// TIA Portal V17 export
// export: Created 2025-03-05T08:03:15.5242576Z, ExportSetting WithDefaults, DisplayName Totally Integrated Automation Portal, DisplayVersion V17 Update 8, DisplayName TIA Portal Openness, DisplayVersion V17 Update 8, DisplayName TIA Portal Version Control Interface, DisplayVersion V17, DisplayName SINAMICS Startdrive Advanced, DisplayVersion V17 SP2, DisplayName SINAMICS Startdrive G110M, G120, G120C, G120D, G120P, G115D, DisplayVersion V17 SP2, DisplayName SINAMICS Startdrive G130, G150, S120, S150, SINAMICS MV, S210, DisplayVersion V17 SP2, DisplayName STEP 7 Professional, DisplayVersion V17 Update 8, DisplayName SINUMERIK ONE STEP 7 Toolbox, DisplayVersion V17 Update 12, DisplayName SINUMERIK 840D sl STEP 7 Toolbox, DisplayVersion V17 Update 12, DisplayName STEP 7 Safety, DisplayVersion V17 Update 6, DisplayName WinCC Advanced, DisplayVersion V17 Update 8
FUNCTION_BLOCK "FB22500_PRESSURE_CONTROL_REGTONIC"   // FB22500, LAD
{ S7_Optimized_Access := 'FALSE' }
VERSION : 0.1
// stored: AutoNumber false, IsIECCheckEnabled false, SetENOAutomatically false, UDAEnableTagReadback false
   VAR_INPUT
      CONTROL_ON_DELAYED : Bool;   // CONTROL ON DELAYED
      PNEUMATIC_CONDITIONS : Bool;   // PNEUMATIC CONDITIONS
      FEEDER_NOT_READY_FAULT : Bool;   // FEEDER NOT READY FAULT
      PRESSURIZE_VALVE_FEEDBACK : Bool;   // PRESSURIZE VALVE FEEDBACK
      START_PROGRAM_REQUEST : Bool;   // START PROGRAM REQUEST
      START_MANUAL_REQUEST : Bool;   // START MANUAL REQUEST
      START_SEMI_REQUEST : Bool;   // START SEMI REQUEST
      START_AUTO_REQUEST : Bool;   // START AUTO REQUEST
      STOP_PROGRAM_REQUEST : Bool;   // STOP PROGRAM REQUEST
      STOP_MANUAL_REQUEST : Bool;   // STOP MANUAL REQUEST
      STOP_SEMI_REQUEST : Bool;   // STOP SEMI REQUEST
      STOP_AUTO_REQUEST : Bool;   // STOP AUTO REQUEST
      ACTUAL_PRESSURE : Real;   // ACTUAL PRESSURE
      PRESSURE_SETPOINT_AUTO : Real;   // PRESSURE SETPOINT
   END_VAR
   VAR_OUTPUT
      PRESSURE_CONTROL_VALUE : Int;   // PRESSURE CONTROL VALUE
      SIMULTANEITY_ALARM : Bool;   // SIMULTANEITY ALARM
      TIME_EXCEEDED_ALARM : Bool;   // TIME EXCEEDED ALARM
      SWITCH_ON_ALARM : Bool;   // SWITCH ON ALARM
      SWITCH_OFF_ALARM : Bool;   // SWITCH OFF ALARM
   END_VAR
   VAR_IN_OUT
      DB_PID : PID_Compact;
   END_VAR
   VAR DB_SPECIFIC
      DATA_STANDARD : "GENERAL_DATA_START_STOP";
      START_STOP_HMI { S7_SetPoint := 'True'} : "HMI_DATA_START_STOP";
      INPUT_SETINGS : Struct
         UNIT_NUMBER : Int;
         HOPPER_NUMBER : Int;
      END_STRUCT;
      DATA_HMI : Struct
         PRESSURE_SETPOINT_VALUE : Real;
      END_STRUCT;
      ALARM_SETINGS : Struct
         TIMER_SIMULTANEITY : TON_TIME;   // SIMULTANEITY TIMER
         TIMER_TIME_EXCEEDED { S7_SetPoint := 'True'} : TON_TIME;
      END_STRUCT;
      SETPOINT_PRESSURE : Real;
      CONTROL_PRESSURE_OUTPUT : Int;
   END_VAR
   VAR_TEMP
      DB_NUMBER : DInt;
      RETVAL : Int;
   END_VAR
   // ALARM_SETINGS.TIMER_SIMULTANEITY.PT := T#100ms;
   // ALARM_SETINGS.TIMER_TIME_EXCEEDED.PT := T#4s;
   VAR_TEMP   // added for the SCL form of the ladder/FBD networks
      _w1 : Bool;
      _w2 : Bool;
   END_VAR
BEGIN

NETWORK
TITLE = READ INSTANCE DB NUMBER
      L     DINO;
      +     10#800000;
      T     #DB_NUMBER;



REGION Network 2: GENERAL CONDITIONS START
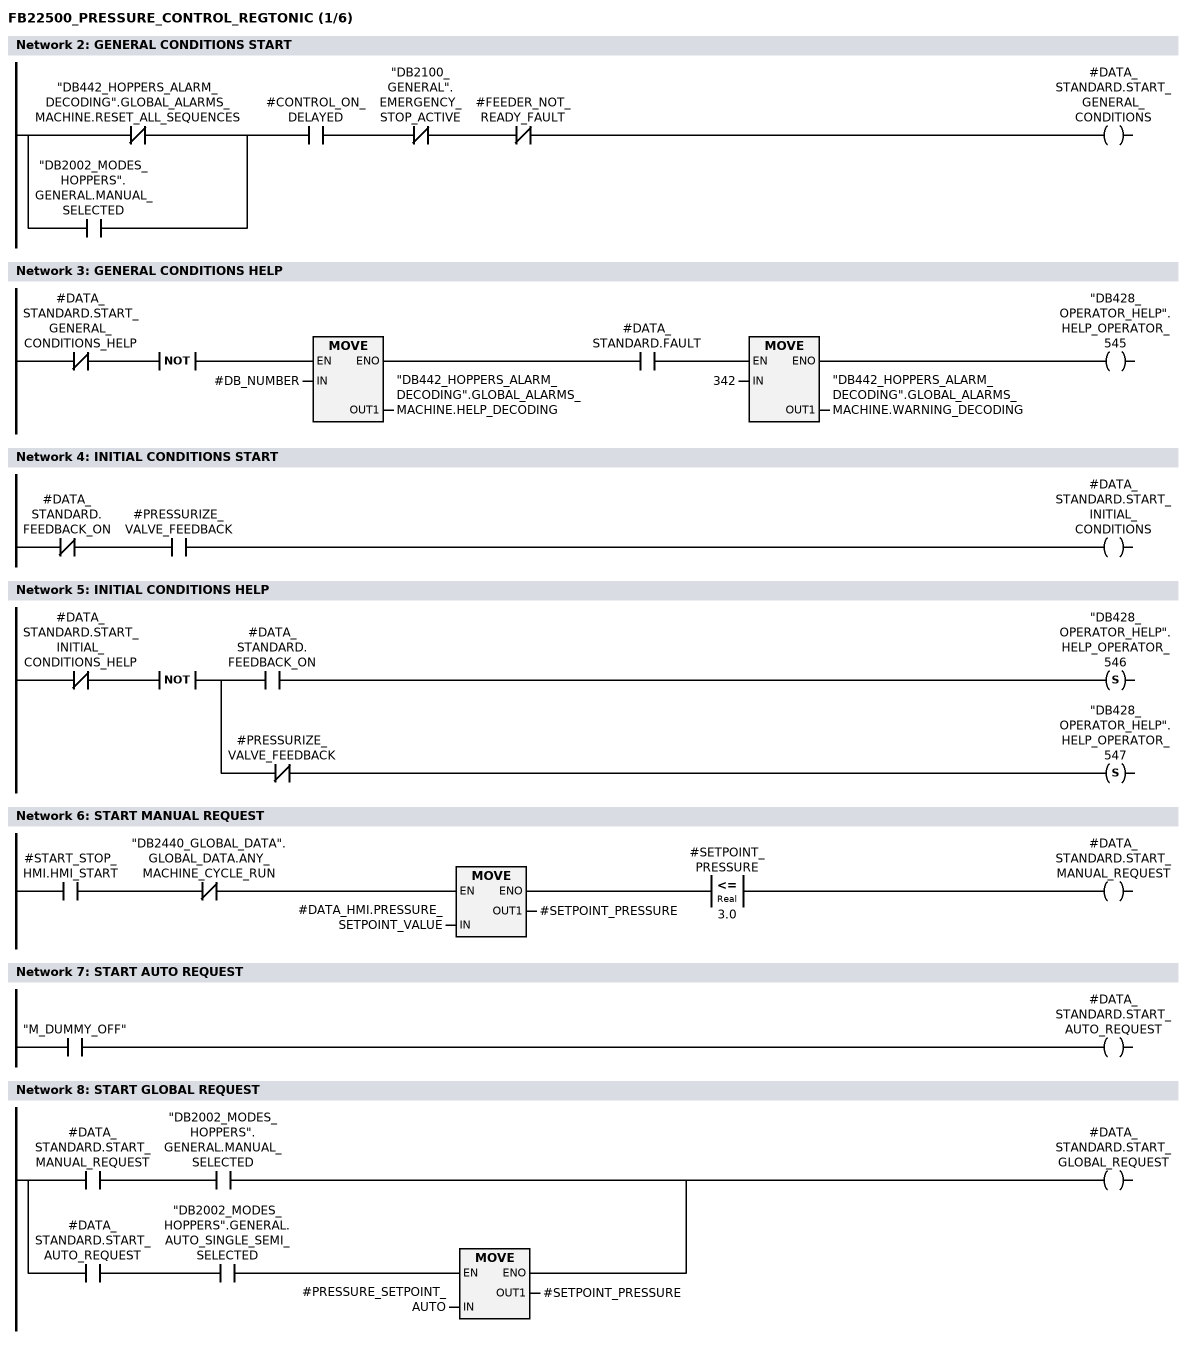
   RUNG wire#powerrail
      I_Contact( "DB442_HOPPERS_ALARM_DECODING".GLOBAL_ALARMS_MACHINE.RESET_ALL_SEQUENCES )
      wire#w1
      Contact( #CONTROL_ON_DELAYED )
      I_Contact( "DB2100_GENERAL".EMERGENCY_STOP_ACTIVE )
      I_Contact( #FEEDER_NOT_READY_FAULT )
      Coil( #DATA_STANDARD.START_GENERAL_CONDITIONS )
   END_RUNG
   RUNG wire#powerrail
      Contact( "DB2002_MODES_HOPPERS".GENERAL.MANUAL_SELECTED )
   END_RUNG wire#w1
   // the same network as SCL:
   #DATA_STANDARD.START_GENERAL_CONDITIONS := (NOT "DB442_HOPPERS_ALARM_DECODING".GLOBAL_ALARMS_MACHINE.RESET_ALL_SEQUENCES OR "DB2002_MODES_HOPPERS".GENERAL.MANUAL_SELECTED) AND #CONTROL_ON_DELAYED AND NOT "DB2100_GENERAL".EMERGENCY_STOP_ACTIVE AND NOT #FEEDER_NOT_READY_FAULT;
END_REGION

REGION Network 3: GENERAL CONDITIONS HELP
   RUNG wire#powerrail
      I_Contact( #DATA_STANDARD.START_GENERAL_CONDITIONS_HELP )
      Not()
      Move(in := #DB_NUMBER, out1 => "DB442_HOPPERS_ALARM_DECODING".GLOBAL_ALARMS_MACHINE.HELP_DECODING)
      Contact( #DATA_STANDARD.FAULT )
      Move(in := 342, out1 => "DB442_HOPPERS_ALARM_DECODING".GLOBAL_ALARMS_MACHINE.WARNING_DECODING)
      Coil( "DB428_OPERATOR_HELP".HELP_OPERATOR_545 )
   END_RUNG
   // the same network as SCL:
   #_w1 := NOT (NOT #DATA_STANDARD.START_GENERAL_CONDITIONS_HELP);
   IF #_w1 THEN "DB442_HOPPERS_ALARM_DECODING".GLOBAL_ALARMS_MACHINE.HELP_DECODING := #DB_NUMBER; END_IF;
   #_w2 := #_w1 AND #DATA_STANDARD.FAULT;
   IF #_w2 THEN "DB442_HOPPERS_ALARM_DECODING".GLOBAL_ALARMS_MACHINE.WARNING_DECODING := 342; END_IF;
   "DB428_OPERATOR_HELP".HELP_OPERATOR_545 := #_w2;
END_REGION

REGION Network 4: INITIAL CONDITIONS START
   RUNG wire#powerrail
      I_Contact( #DATA_STANDARD.FEEDBACK_ON )
      Contact( #PRESSURIZE_VALVE_FEEDBACK )
      Coil( #DATA_STANDARD.START_INITIAL_CONDITIONS )
   END_RUNG
   // the same network as SCL:
   #DATA_STANDARD.START_INITIAL_CONDITIONS := NOT #DATA_STANDARD.FEEDBACK_ON AND #PRESSURIZE_VALVE_FEEDBACK;
END_REGION

REGION Network 5: INITIAL CONDITIONS HELP
   RUNG wire#powerrail
      I_Contact( #DATA_STANDARD.START_INITIAL_CONDITIONS_HELP )
      Not()
      wire#w1
      Contact( #DATA_STANDARD.FEEDBACK_ON )
      S_Coil( "DB428_OPERATOR_HELP".HELP_OPERATOR_546 )
   END_RUNG
   RUNG wire#w1
      I_Contact( #PRESSURIZE_VALVE_FEEDBACK )
      S_Coil( "DB428_OPERATOR_HELP".HELP_OPERATOR_547 )
   END_RUNG
   // the same network as SCL:
   #_w1 := NOT (NOT #DATA_STANDARD.START_INITIAL_CONDITIONS_HELP);
   IF #_w1 AND #DATA_STANDARD.FEEDBACK_ON THEN "DB428_OPERATOR_HELP".HELP_OPERATOR_546 := TRUE; END_IF;
   IF #_w1 AND NOT #PRESSURIZE_VALVE_FEEDBACK THEN "DB428_OPERATOR_HELP".HELP_OPERATOR_547 := TRUE; END_IF;
END_REGION

REGION Network 6: START MANUAL REQUEST
   RUNG wire#powerrail
      Contact( #START_STOP_HMI.HMI_START )
      I_Contact( "DB2440_GLOBAL_DATA".GLOBAL_DATA.ANY_MACHINE_CYCLE_RUN )
      Move(in := #DATA_HMI.PRESSURE_SETPOINT_VALUE, out1 => #SETPOINT_PRESSURE)
      { S7_Templates := "SrcType := Real" } LE_Contact(in1 := #SETPOINT_PRESSURE, in2 := 3.0)
      Coil( #DATA_STANDARD.START_MANUAL_REQUEST )
   END_RUNG
   // the same network as SCL:
   #_w1 := #START_STOP_HMI.HMI_START AND NOT "DB2440_GLOBAL_DATA".GLOBAL_DATA.ANY_MACHINE_CYCLE_RUN;
   IF #_w1 THEN #SETPOINT_PRESSURE := #DATA_HMI.PRESSURE_SETPOINT_VALUE; END_IF;
   #DATA_STANDARD.START_MANUAL_REQUEST := #_w1 AND (#SETPOINT_PRESSURE <= 3.0);
END_REGION

REGION Network 7: START AUTO REQUEST
   RUNG wire#powerrail
      Contact( "M_DUMMY_OFF" )
      Coil( #DATA_STANDARD.START_AUTO_REQUEST )
   END_RUNG
   // the same network as SCL:
   #DATA_STANDARD.START_AUTO_REQUEST := "M_DUMMY_OFF";
END_REGION

REGION Network 8: START GLOBAL REQUEST
   RUNG wire#powerrail
      Contact( #DATA_STANDARD.START_MANUAL_REQUEST )
      Contact( "DB2002_MODES_HOPPERS".GENERAL.MANUAL_SELECTED )
      wire#w1
      Coil( #DATA_STANDARD.START_GLOBAL_REQUEST )
   END_RUNG
   RUNG wire#powerrail
      Contact( #DATA_STANDARD.START_AUTO_REQUEST )
      Contact( "DB2002_MODES_HOPPERS".GENERAL.AUTO_SINGLE_SEMI_SELECTED )
      Move(in := #PRESSURE_SETPOINT_AUTO, out1 => #SETPOINT_PRESSURE)
   END_RUNG wire#w1
   // the same network as SCL:
   #_w1 := #DATA_STANDARD.START_AUTO_REQUEST AND "DB2002_MODES_HOPPERS".GENERAL.AUTO_SINGLE_SEMI_SELECTED;
   IF #_w1 THEN #SETPOINT_PRESSURE := #PRESSURE_SETPOINT_AUTO; END_IF;
   #DATA_STANDARD.START_GLOBAL_REQUEST := (#DATA_STANDARD.START_MANUAL_REQUEST AND "DB2002_MODES_HOPPERS".GENERAL.MANUAL_SELECTED) OR #_w1;
END_REGION

REGION Network 9: START COMMAND
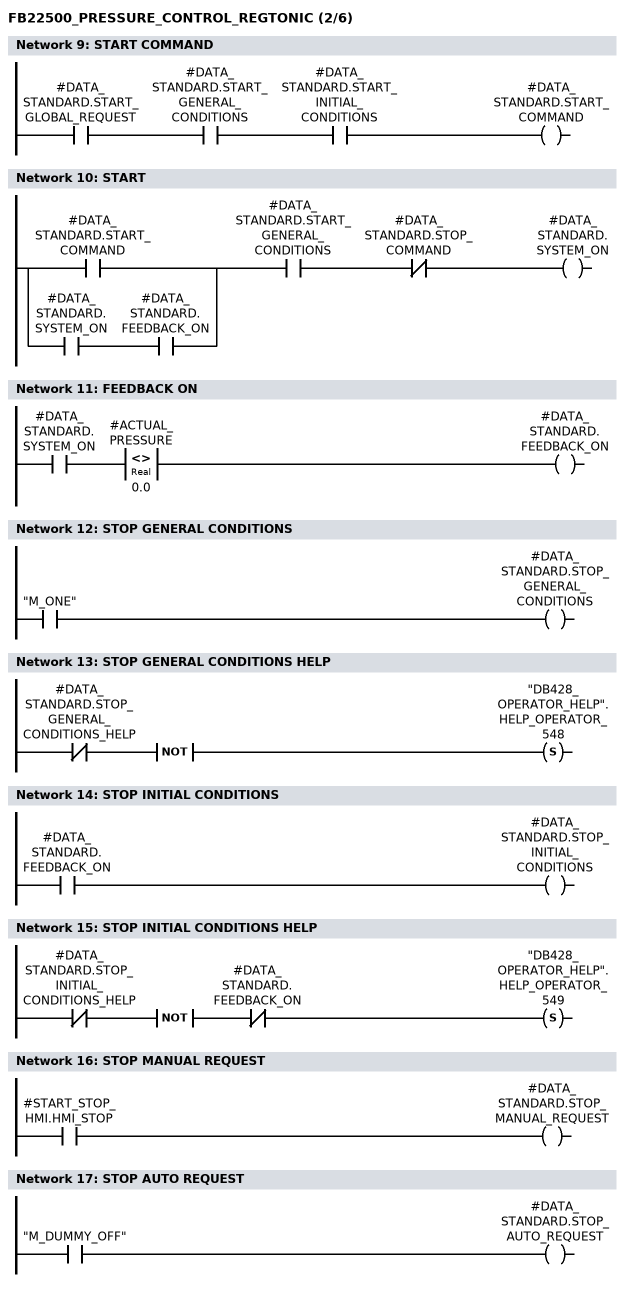
   RUNG wire#powerrail
      Contact( #DATA_STANDARD.START_GLOBAL_REQUEST )
      Contact( #DATA_STANDARD.START_GENERAL_CONDITIONS )
      Contact( #DATA_STANDARD.START_INITIAL_CONDITIONS )
      Coil( #DATA_STANDARD.START_COMMAND )
   END_RUNG
   // the same network as SCL:
   #DATA_STANDARD.START_COMMAND := #DATA_STANDARD.START_GLOBAL_REQUEST AND #DATA_STANDARD.START_GENERAL_CONDITIONS AND #DATA_STANDARD.START_INITIAL_CONDITIONS;
END_REGION

REGION Network 10: START
   RUNG wire#powerrail
      Contact( #DATA_STANDARD.START_COMMAND )
      wire#w1
      Contact( #DATA_STANDARD.START_GENERAL_CONDITIONS )
      I_Contact( #DATA_STANDARD.STOP_COMMAND )
      Coil( #DATA_STANDARD.SYSTEM_ON )
   END_RUNG
   RUNG wire#powerrail
      Contact( #DATA_STANDARD.SYSTEM_ON )
      Contact( #DATA_STANDARD.FEEDBACK_ON )
   END_RUNG wire#w1
   // the same network as SCL:
   #DATA_STANDARD.SYSTEM_ON := (#DATA_STANDARD.START_COMMAND OR (#DATA_STANDARD.SYSTEM_ON AND #DATA_STANDARD.FEEDBACK_ON)) AND #DATA_STANDARD.START_GENERAL_CONDITIONS AND NOT #DATA_STANDARD.STOP_COMMAND;
END_REGION

REGION Network 11: FEEDBACK ON
   RUNG wire#powerrail
      Contact( #DATA_STANDARD.SYSTEM_ON )
      { S7_Templates := "SrcType := Real" } NE_Contact(in1 := #ACTUAL_PRESSURE, in2 := 0.0)
      Coil( #DATA_STANDARD.FEEDBACK_ON )
   END_RUNG
   // the same network as SCL:
   #DATA_STANDARD.FEEDBACK_ON := #DATA_STANDARD.SYSTEM_ON AND (#ACTUAL_PRESSURE <> 0.0);
END_REGION

REGION Network 12: STOP GENERAL CONDITIONS
   RUNG wire#powerrail
      Contact( "M_ONE" )
      Coil( #DATA_STANDARD.STOP_GENERAL_CONDITIONS )
   END_RUNG
   // the same network as SCL:
   #DATA_STANDARD.STOP_GENERAL_CONDITIONS := "M_ONE";
END_REGION

REGION Network 13: STOP GENERAL CONDITIONS HELP
   RUNG wire#powerrail
      I_Contact( #DATA_STANDARD.STOP_GENERAL_CONDITIONS_HELP )
      Not()
      S_Coil( "DB428_OPERATOR_HELP".HELP_OPERATOR_548 )
   END_RUNG
   // the same network as SCL:
   IF NOT (NOT #DATA_STANDARD.STOP_GENERAL_CONDITIONS_HELP) THEN
       "DB428_OPERATOR_HELP".HELP_OPERATOR_548 := TRUE;
   END_IF;
END_REGION

REGION Network 14: STOP INITIAL CONDITIONS
   RUNG wire#powerrail
      Contact( #DATA_STANDARD.FEEDBACK_ON )
      Coil( #DATA_STANDARD.STOP_INITIAL_CONDITIONS )
   END_RUNG
   // the same network as SCL:
   #DATA_STANDARD.STOP_INITIAL_CONDITIONS := #DATA_STANDARD.FEEDBACK_ON;
END_REGION

REGION Network 15: STOP INITIAL CONDITIONS HELP
   RUNG wire#powerrail
      I_Contact( #DATA_STANDARD.STOP_INITIAL_CONDITIONS_HELP )
      Not()
      I_Contact( #DATA_STANDARD.FEEDBACK_ON )
      S_Coil( "DB428_OPERATOR_HELP".HELP_OPERATOR_549 )
   END_RUNG
   // the same network as SCL:
   IF NOT (NOT #DATA_STANDARD.STOP_INITIAL_CONDITIONS_HELP) AND NOT #DATA_STANDARD.FEEDBACK_ON THEN
       "DB428_OPERATOR_HELP".HELP_OPERATOR_549 := TRUE;
   END_IF;
END_REGION

REGION Network 16: STOP MANUAL REQUEST
   RUNG wire#powerrail
      Contact( #START_STOP_HMI.HMI_STOP )
      Coil( #DATA_STANDARD.STOP_MANUAL_REQUEST )
   END_RUNG
   // the same network as SCL:
   #DATA_STANDARD.STOP_MANUAL_REQUEST := #START_STOP_HMI.HMI_STOP;
END_REGION

REGION Network 17: STOP AUTO REQUEST
   RUNG wire#powerrail
      Contact( "M_DUMMY_OFF" )
      Coil( #DATA_STANDARD.STOP_AUTO_REQUEST )
   END_RUNG
   // the same network as SCL:
   #DATA_STANDARD.STOP_AUTO_REQUEST := "M_DUMMY_OFF";
END_REGION

REGION Network 18: STOP GLOBAL REQUEST
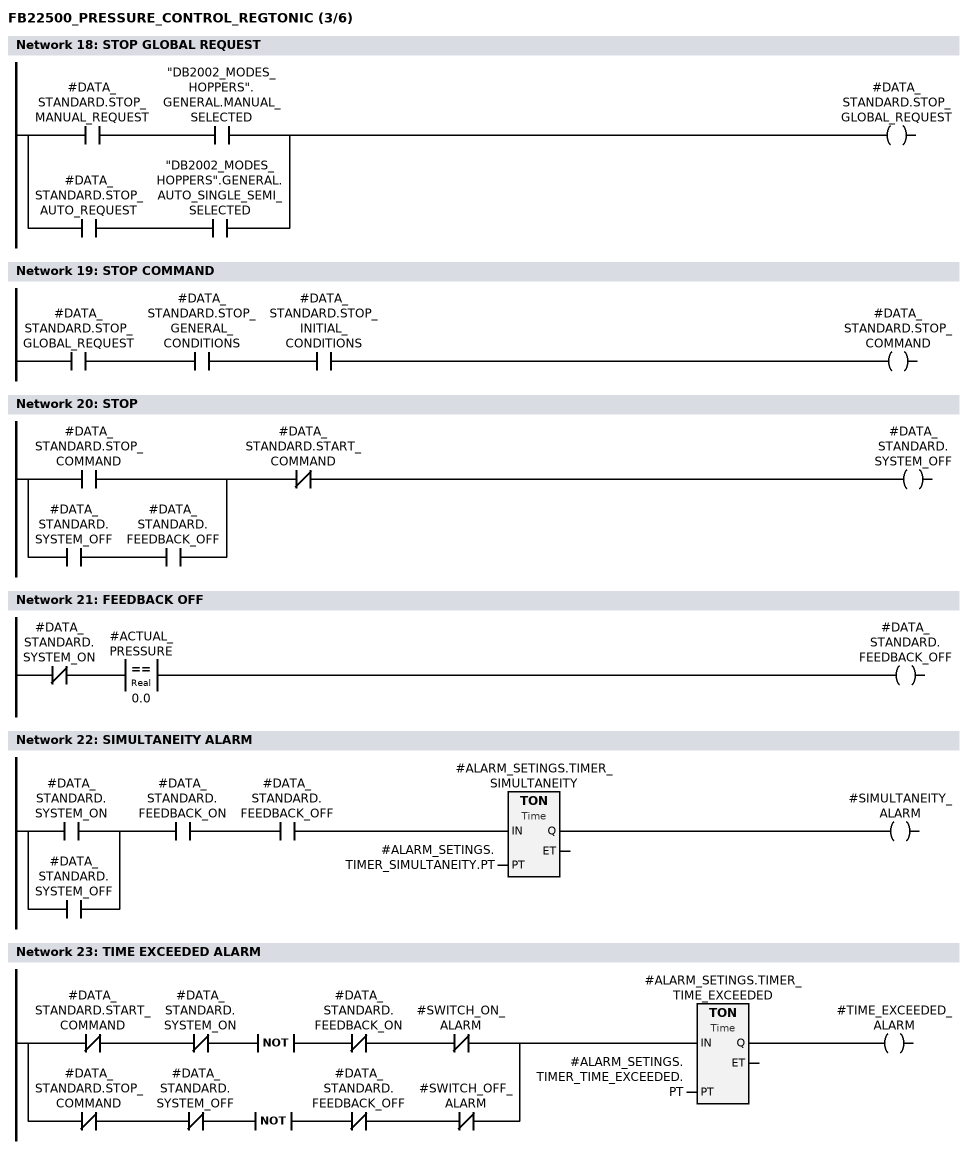
   RUNG wire#powerrail
      Contact( #DATA_STANDARD.STOP_MANUAL_REQUEST )
      Contact( "DB2002_MODES_HOPPERS".GENERAL.MANUAL_SELECTED )
      wire#w1
      Coil( #DATA_STANDARD.STOP_GLOBAL_REQUEST )
   END_RUNG
   RUNG wire#powerrail
      Contact( #DATA_STANDARD.STOP_AUTO_REQUEST )
      Contact( "DB2002_MODES_HOPPERS".GENERAL.AUTO_SINGLE_SEMI_SELECTED )
   END_RUNG wire#w1
   // the same network as SCL:
   #DATA_STANDARD.STOP_GLOBAL_REQUEST := (#DATA_STANDARD.STOP_MANUAL_REQUEST AND "DB2002_MODES_HOPPERS".GENERAL.MANUAL_SELECTED) OR (#DATA_STANDARD.STOP_AUTO_REQUEST AND "DB2002_MODES_HOPPERS".GENERAL.AUTO_SINGLE_SEMI_SELECTED);
END_REGION

REGION Network 19: STOP COMMAND
   RUNG wire#powerrail
      Contact( #DATA_STANDARD.STOP_GLOBAL_REQUEST )
      Contact( #DATA_STANDARD.STOP_GENERAL_CONDITIONS )
      Contact( #DATA_STANDARD.STOP_INITIAL_CONDITIONS )
      Coil( #DATA_STANDARD.STOP_COMMAND )
   END_RUNG
   // the same network as SCL:
   #DATA_STANDARD.STOP_COMMAND := #DATA_STANDARD.STOP_GLOBAL_REQUEST AND #DATA_STANDARD.STOP_GENERAL_CONDITIONS AND #DATA_STANDARD.STOP_INITIAL_CONDITIONS;
END_REGION

REGION Network 20: STOP
   RUNG wire#powerrail
      Contact( #DATA_STANDARD.STOP_COMMAND )
      wire#w1
      I_Contact( #DATA_STANDARD.START_COMMAND )
      Coil( #DATA_STANDARD.SYSTEM_OFF )
   END_RUNG
   RUNG wire#powerrail
      Contact( #DATA_STANDARD.SYSTEM_OFF )
      Contact( #DATA_STANDARD.FEEDBACK_OFF )
   END_RUNG wire#w1
   // the same network as SCL:
   #DATA_STANDARD.SYSTEM_OFF := (#DATA_STANDARD.STOP_COMMAND OR (#DATA_STANDARD.SYSTEM_OFF AND #DATA_STANDARD.FEEDBACK_OFF)) AND NOT #DATA_STANDARD.START_COMMAND;
END_REGION

REGION Network 21: FEEDBACK OFF
   RUNG wire#powerrail
      I_Contact( #DATA_STANDARD.SYSTEM_ON )
      { S7_Templates := "SrcType := Real" } EQ_Contact(in1 := #ACTUAL_PRESSURE, in2 := 0.0)
      Coil( #DATA_STANDARD.FEEDBACK_OFF )
   END_RUNG
   // the same network as SCL:
   #DATA_STANDARD.FEEDBACK_OFF := NOT #DATA_STANDARD.SYSTEM_ON AND (#ACTUAL_PRESSURE = 0.0);
END_REGION

REGION Network 22: SIMULTANEITY ALARM
   RUNG wire#powerrail
      Contact( #DATA_STANDARD.SYSTEM_ON )
      wire#w1
      Contact( #DATA_STANDARD.FEEDBACK_ON )
      Contact( #DATA_STANDARD.FEEDBACK_OFF )
      { S7_Templates := "time_type := Time" } #ALARM_SETINGS.TIMER_SIMULTANEITY.TON(pt := #ALARM_SETINGS.TIMER_SIMULTANEITY.PT, et =>)
      Coil( #SIMULTANEITY_ALARM )
   END_RUNG
   RUNG wire#powerrail
      Contact( #DATA_STANDARD.SYSTEM_OFF )
   END_RUNG wire#w1
   // the same network as SCL:
   #ALARM_SETINGS.TIMER_SIMULTANEITY.TON(IN := (#DATA_STANDARD.SYSTEM_ON OR #DATA_STANDARD.SYSTEM_OFF) AND #DATA_STANDARD.FEEDBACK_ON AND #DATA_STANDARD.FEEDBACK_OFF,
                           PT := #ALARM_SETINGS.TIMER_SIMULTANEITY.PT);
   #SIMULTANEITY_ALARM := #ALARM_SETINGS.TIMER_SIMULTANEITY.Q;
END_REGION

REGION Network 23: TIME EXCEEDED ALARM
   RUNG wire#powerrail
      I_Contact( #DATA_STANDARD.START_COMMAND )
      I_Contact( #DATA_STANDARD.SYSTEM_ON )
      Not()
      I_Contact( #DATA_STANDARD.FEEDBACK_ON )
      I_Contact( #SWITCH_ON_ALARM )
      wire#w1
      { S7_Templates := "time_type := Time" } #ALARM_SETINGS.TIMER_TIME_EXCEEDED.TON(pt := #ALARM_SETINGS.TIMER_TIME_EXCEEDED.PT, et =>)
      Coil( #TIME_EXCEEDED_ALARM )
   END_RUNG
   RUNG wire#powerrail
      I_Contact( #DATA_STANDARD.STOP_COMMAND )
      I_Contact( #DATA_STANDARD.SYSTEM_OFF )
      Not()
      I_Contact( #DATA_STANDARD.FEEDBACK_OFF )
      I_Contact( #SWITCH_OFF_ALARM )
   END_RUNG wire#w1
   // the same network as SCL:
   #ALARM_SETINGS.TIMER_TIME_EXCEEDED.TON(IN := (NOT (NOT #DATA_STANDARD.START_COMMAND AND NOT #DATA_STANDARD.SYSTEM_ON) AND NOT #DATA_STANDARD.FEEDBACK_ON AND NOT #SWITCH_ON_ALARM) OR (NOT (NOT #DATA_STANDARD.STOP_COMMAND AND NOT #DATA_STANDARD.SYSTEM_OFF) AND NOT #DATA_STANDARD.FEEDBACK_OFF AND NOT #SWITCH_OFF_ALARM),
                           PT := #ALARM_SETINGS.TIMER_TIME_EXCEEDED.PT);
   #TIME_EXCEEDED_ALARM := #ALARM_SETINGS.TIMER_TIME_EXCEEDED.Q;
END_REGION

REGION Network 24: SWITCH ON ALARM
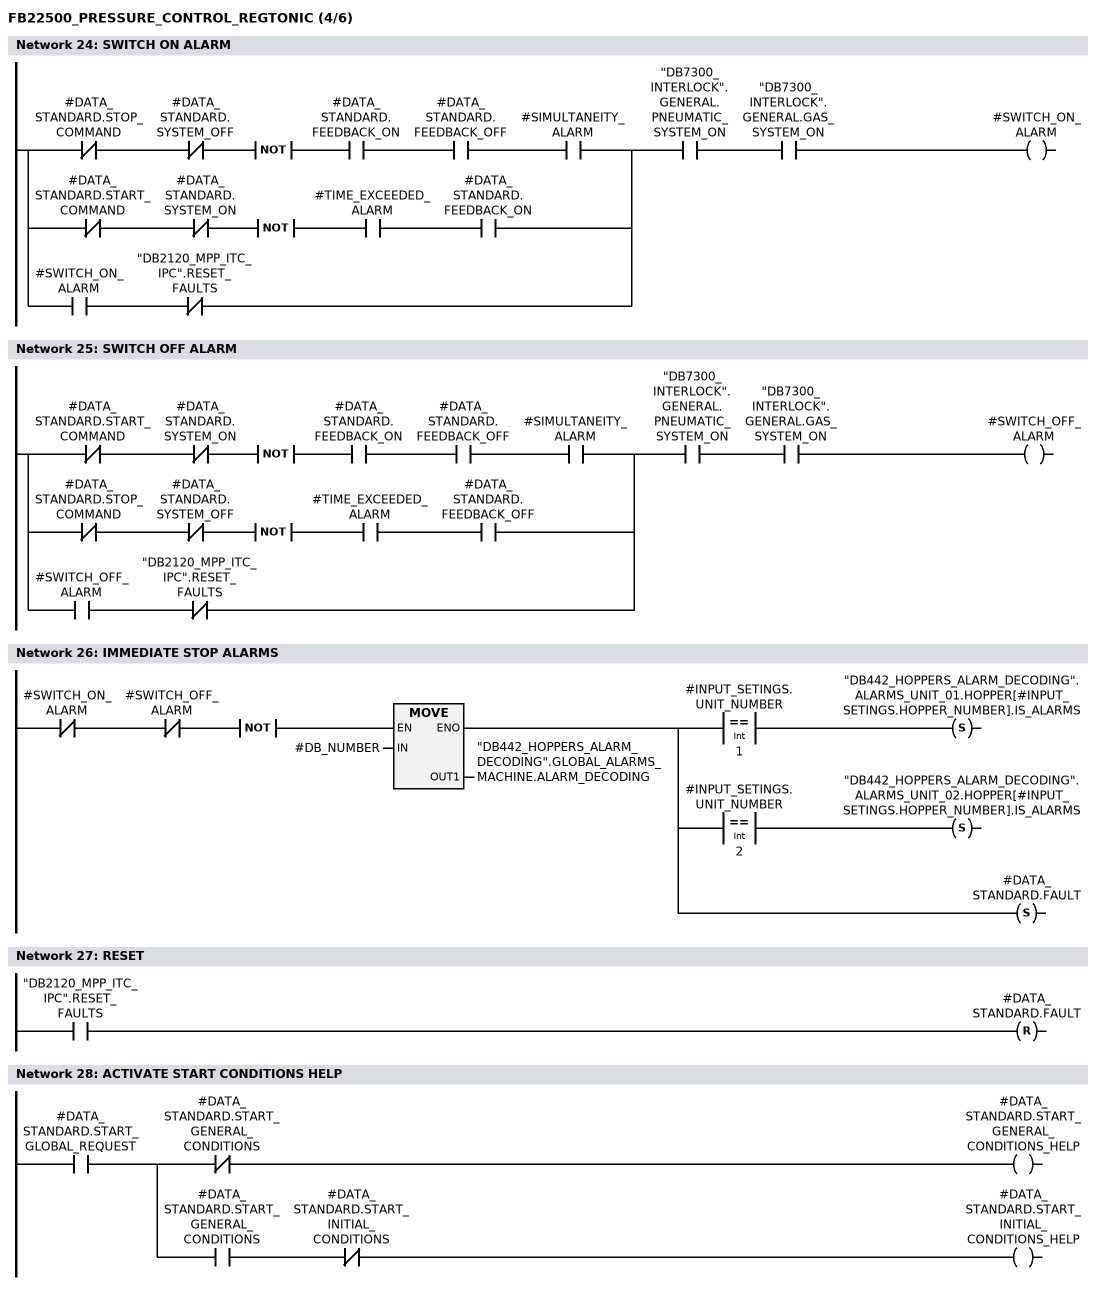
   RUNG wire#powerrail
      I_Contact( #DATA_STANDARD.STOP_COMMAND )
      I_Contact( #DATA_STANDARD.SYSTEM_OFF )
      Not()
      Contact( #DATA_STANDARD.FEEDBACK_ON )
      Contact( #DATA_STANDARD.FEEDBACK_OFF )
      Contact( #SIMULTANEITY_ALARM )
      wire#w1
      Contact( "DB7300_INTERLOCK".GENERAL.PNEUMATIC_SYSTEM_ON )
      Contact( "DB7300_INTERLOCK".GENERAL.GAS_SYSTEM_ON )
      Coil( #SWITCH_ON_ALARM )
   END_RUNG
   RUNG wire#powerrail
      I_Contact( #DATA_STANDARD.START_COMMAND )
      I_Contact( #DATA_STANDARD.SYSTEM_ON )
      Not()
      Contact( #TIME_EXCEEDED_ALARM )
      Contact( #DATA_STANDARD.FEEDBACK_ON )
   END_RUNG wire#w1
   RUNG wire#powerrail
      Contact( #SWITCH_ON_ALARM )
      I_Contact( "DB2120_MPP_ITC_IPC".RESET_FAULTS )
   END_RUNG wire#w1
   // the same network as SCL:
   #SWITCH_ON_ALARM := ((NOT (NOT #DATA_STANDARD.STOP_COMMAND AND NOT #DATA_STANDARD.SYSTEM_OFF) AND #DATA_STANDARD.FEEDBACK_ON AND #DATA_STANDARD.FEEDBACK_OFF AND #SIMULTANEITY_ALARM) OR (NOT (NOT #DATA_STANDARD.START_COMMAND AND NOT #DATA_STANDARD.SYSTEM_ON) AND #TIME_EXCEEDED_ALARM AND #DATA_STANDARD.FEEDBACK_ON) OR (#SWITCH_ON_ALARM AND NOT "DB2120_MPP_ITC_IPC".RESET_FAULTS)) AND "DB7300_INTERLOCK".GENERAL.PNEUMATIC_SYSTEM_ON AND "DB7300_INTERLOCK".GENERAL.GAS_SYSTEM_ON;
END_REGION

REGION Network 25: SWITCH OFF ALARM
   RUNG wire#powerrail
      I_Contact( #DATA_STANDARD.START_COMMAND )
      I_Contact( #DATA_STANDARD.SYSTEM_ON )
      Not()
      Contact( #DATA_STANDARD.FEEDBACK_ON )
      Contact( #DATA_STANDARD.FEEDBACK_OFF )
      Contact( #SIMULTANEITY_ALARM )
      wire#w1
      Contact( "DB7300_INTERLOCK".GENERAL.PNEUMATIC_SYSTEM_ON )
      Contact( "DB7300_INTERLOCK".GENERAL.GAS_SYSTEM_ON )
      Coil( #SWITCH_OFF_ALARM )
   END_RUNG
   RUNG wire#powerrail
      I_Contact( #DATA_STANDARD.STOP_COMMAND )
      I_Contact( #DATA_STANDARD.SYSTEM_OFF )
      Not()
      Contact( #TIME_EXCEEDED_ALARM )
      Contact( #DATA_STANDARD.FEEDBACK_OFF )
   END_RUNG wire#w1
   RUNG wire#powerrail
      Contact( #SWITCH_OFF_ALARM )
      I_Contact( "DB2120_MPP_ITC_IPC".RESET_FAULTS )
   END_RUNG wire#w1
   // the same network as SCL:
   #SWITCH_OFF_ALARM := ((NOT (NOT #DATA_STANDARD.START_COMMAND AND NOT #DATA_STANDARD.SYSTEM_ON) AND #DATA_STANDARD.FEEDBACK_ON AND #DATA_STANDARD.FEEDBACK_OFF AND #SIMULTANEITY_ALARM) OR (NOT (NOT #DATA_STANDARD.STOP_COMMAND AND NOT #DATA_STANDARD.SYSTEM_OFF) AND #TIME_EXCEEDED_ALARM AND #DATA_STANDARD.FEEDBACK_OFF) OR (#SWITCH_OFF_ALARM AND NOT "DB2120_MPP_ITC_IPC".RESET_FAULTS)) AND "DB7300_INTERLOCK".GENERAL.PNEUMATIC_SYSTEM_ON AND "DB7300_INTERLOCK".GENERAL.GAS_SYSTEM_ON;
END_REGION

REGION Network 26: IMMEDIATE STOP ALARMS
   RUNG wire#powerrail
      I_Contact( #SWITCH_ON_ALARM )
      I_Contact( #SWITCH_OFF_ALARM )
      Not()
      Move(in := #DB_NUMBER, out1 => "DB442_HOPPERS_ALARM_DECODING".GLOBAL_ALARMS_MACHINE.ALARM_DECODING)
      wire#w1
      { S7_Templates := "SrcType := Int" } EQ_Contact(in1 := #INPUT_SETINGS.UNIT_NUMBER, in2 := 1)
      S_Coil( "DB442_HOPPERS_ALARM_DECODING".ALARMS_UNIT_01.HOPPER[#INPUT_SETINGS.HOPPER_NUMBER].IS_ALARMS )
   END_RUNG
   RUNG wire#w1
      { S7_Templates := "SrcType := Int" } EQ_Contact(in1 := #INPUT_SETINGS.UNIT_NUMBER, in2 := 2)
      S_Coil( "DB442_HOPPERS_ALARM_DECODING".ALARMS_UNIT_02.HOPPER[#INPUT_SETINGS.HOPPER_NUMBER].IS_ALARMS )
   END_RUNG
   RUNG wire#w1
      S_Coil( #DATA_STANDARD.FAULT )
   END_RUNG
   // the same network as SCL:
   #_w1 := NOT (NOT #SWITCH_ON_ALARM AND NOT #SWITCH_OFF_ALARM);
   IF #_w1 THEN "DB442_HOPPERS_ALARM_DECODING".GLOBAL_ALARMS_MACHINE.ALARM_DECODING := #DB_NUMBER; END_IF;
   IF #_w1 AND (#INPUT_SETINGS.UNIT_NUMBER = 1) THEN
       "DB442_HOPPERS_ALARM_DECODING".ALARMS_UNIT_01.HOPPER[#INPUT_SETINGS.HOPPER_NUMBER].IS_ALARMS := TRUE;
   END_IF;
   IF #_w1 AND (#INPUT_SETINGS.UNIT_NUMBER = 2) THEN
       "DB442_HOPPERS_ALARM_DECODING".ALARMS_UNIT_02.HOPPER[#INPUT_SETINGS.HOPPER_NUMBER].IS_ALARMS := TRUE;
   END_IF;
   IF #_w1 THEN #DATA_STANDARD.FAULT := TRUE; END_IF;
END_REGION

REGION Network 27: RESET
   RUNG wire#powerrail
      Contact( "DB2120_MPP_ITC_IPC".RESET_FAULTS )
      R_Coil( #DATA_STANDARD.FAULT )
   END_RUNG
   // the same network as SCL:
   IF "DB2120_MPP_ITC_IPC".RESET_FAULTS THEN #DATA_STANDARD.FAULT := FALSE; END_IF;
END_REGION

REGION Network 28: ACTIVATE START CONDITIONS HELP
   RUNG wire#powerrail
      Contact( #DATA_STANDARD.START_GLOBAL_REQUEST )
      wire#w1
      I_Contact( #DATA_STANDARD.START_GENERAL_CONDITIONS )
      Coil( #DATA_STANDARD.START_GENERAL_CONDITIONS_HELP )
   END_RUNG
   RUNG wire#w1
      Contact( #DATA_STANDARD.START_GENERAL_CONDITIONS )
      I_Contact( #DATA_STANDARD.START_INITIAL_CONDITIONS )
      Coil( #DATA_STANDARD.START_INITIAL_CONDITIONS_HELP )
   END_RUNG
   // the same network as SCL:
   #DATA_STANDARD.START_GENERAL_CONDITIONS_HELP := #DATA_STANDARD.START_GLOBAL_REQUEST AND NOT #DATA_STANDARD.START_GENERAL_CONDITIONS;
   #DATA_STANDARD.START_INITIAL_CONDITIONS_HELP := #DATA_STANDARD.START_GLOBAL_REQUEST AND #DATA_STANDARD.START_GENERAL_CONDITIONS AND NOT #DATA_STANDARD.START_INITIAL_CONDITIONS;
END_REGION

REGION Network 29: ACTIVATE STOP CONDITIONS HELP
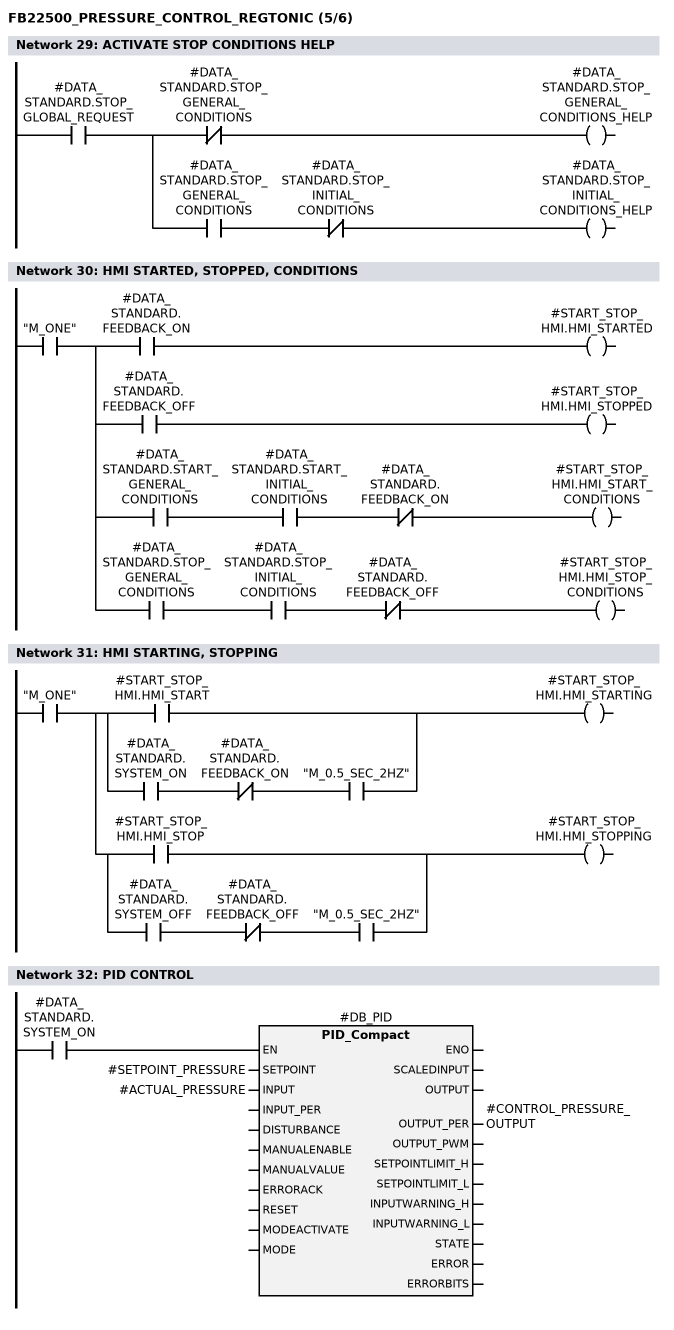
   RUNG wire#powerrail
      Contact( #DATA_STANDARD.STOP_GLOBAL_REQUEST )
      wire#w1
      I_Contact( #DATA_STANDARD.STOP_GENERAL_CONDITIONS )
      Coil( #DATA_STANDARD.STOP_GENERAL_CONDITIONS_HELP )
   END_RUNG
   RUNG wire#w1
      Contact( #DATA_STANDARD.STOP_GENERAL_CONDITIONS )
      I_Contact( #DATA_STANDARD.STOP_INITIAL_CONDITIONS )
      Coil( #DATA_STANDARD.STOP_INITIAL_CONDITIONS_HELP )
   END_RUNG
   // the same network as SCL:
   #DATA_STANDARD.STOP_GENERAL_CONDITIONS_HELP := #DATA_STANDARD.STOP_GLOBAL_REQUEST AND NOT #DATA_STANDARD.STOP_GENERAL_CONDITIONS;
   #DATA_STANDARD.STOP_INITIAL_CONDITIONS_HELP := #DATA_STANDARD.STOP_GLOBAL_REQUEST AND #DATA_STANDARD.STOP_GENERAL_CONDITIONS AND NOT #DATA_STANDARD.STOP_INITIAL_CONDITIONS;
END_REGION

REGION Network 30: HMI STARTED, STOPPED, CONDITIONS
   RUNG wire#powerrail
      Contact( "M_ONE" )
      wire#w1
      Contact( #DATA_STANDARD.FEEDBACK_ON )
      Coil( #START_STOP_HMI.HMI_STARTED )
   END_RUNG
   RUNG wire#w1
      Contact( #DATA_STANDARD.FEEDBACK_OFF )
      Coil( #START_STOP_HMI.HMI_STOPPED )
   END_RUNG
   RUNG wire#w1
      Contact( #DATA_STANDARD.START_GENERAL_CONDITIONS )
      Contact( #DATA_STANDARD.START_INITIAL_CONDITIONS )
      I_Contact( #DATA_STANDARD.FEEDBACK_ON )
      Coil( #START_STOP_HMI.HMI_START_CONDITIONS )
   END_RUNG
   RUNG wire#w1
      Contact( #DATA_STANDARD.STOP_GENERAL_CONDITIONS )
      Contact( #DATA_STANDARD.STOP_INITIAL_CONDITIONS )
      I_Contact( #DATA_STANDARD.FEEDBACK_OFF )
      Coil( #START_STOP_HMI.HMI_STOP_CONDITIONS )
   END_RUNG
   // the same network as SCL:
   #START_STOP_HMI.HMI_STARTED := "M_ONE" AND #DATA_STANDARD.FEEDBACK_ON;
   #START_STOP_HMI.HMI_STOPPED := "M_ONE" AND #DATA_STANDARD.FEEDBACK_OFF;
   #START_STOP_HMI.HMI_START_CONDITIONS := "M_ONE" AND #DATA_STANDARD.START_GENERAL_CONDITIONS AND #DATA_STANDARD.START_INITIAL_CONDITIONS AND NOT #DATA_STANDARD.FEEDBACK_ON;
   #START_STOP_HMI.HMI_STOP_CONDITIONS := "M_ONE" AND #DATA_STANDARD.STOP_GENERAL_CONDITIONS AND #DATA_STANDARD.STOP_INITIAL_CONDITIONS AND NOT #DATA_STANDARD.FEEDBACK_OFF;
END_REGION

REGION Network 31: HMI STARTING, STOPPING
   RUNG wire#powerrail
      Contact( "M_ONE" )
      wire#w1
      Contact( #START_STOP_HMI.HMI_START )
      wire#w2
      Coil( #START_STOP_HMI.HMI_STARTING )
   END_RUNG
   RUNG wire#w1
      Contact( #DATA_STANDARD.SYSTEM_ON )
      I_Contact( #DATA_STANDARD.FEEDBACK_ON )
      Contact( "M_0.5_SEC_2HZ" )
   END_RUNG wire#w2
   RUNG wire#w1
      Contact( #START_STOP_HMI.HMI_STOP )
      wire#w3
      Coil( #START_STOP_HMI.HMI_STOPPING )
   END_RUNG
   RUNG wire#w1
      Contact( #DATA_STANDARD.SYSTEM_OFF )
      I_Contact( #DATA_STANDARD.FEEDBACK_OFF )
      Contact( "M_0.5_SEC_2HZ" )
   END_RUNG wire#w3
   // the same network as SCL:
   #START_STOP_HMI.HMI_STARTING := "M_ONE" AND (#START_STOP_HMI.HMI_START OR (#DATA_STANDARD.SYSTEM_ON AND NOT #DATA_STANDARD.FEEDBACK_ON AND "M_0.5_SEC_2HZ"));
   #START_STOP_HMI.HMI_STOPPING := "M_ONE" AND (#START_STOP_HMI.HMI_STOP OR (#DATA_STANDARD.SYSTEM_OFF AND NOT #DATA_STANDARD.FEEDBACK_OFF AND "M_0.5_SEC_2HZ"));
END_REGION

REGION Network 32: PID CONTROL
   RUNG wire#powerrail
      Contact( #DATA_STANDARD.SYSTEM_ON )
      #DB_PID.PID_Compact(Setpoint := #SETPOINT_PRESSURE, Input := #ACTUAL_PRESSURE, Input_PER :=, Disturbance :=, ManualEnable :=, ManualValue :=, ErrorAck :=, Reset :=, ModeActivate :=, Mode :=, ScaledInput =>, Output =>, Output_PER => #CONTROL_PRESSURE_OUTPUT, Output_PWM =>, SetpointLimit_H =>, SetpointLimit_L =>, InputWarning_H =>, InputWarning_L =>, State =>, Error =>, ErrorBits =>)
   END_RUNG
   // the same network as SCL:
   IF #DATA_STANDARD.SYSTEM_ON THEN
       #DB_PID(Setpoint := #SETPOINT_PRESSURE, Input := #ACTUAL_PRESSURE, Output_PER => #CONTROL_PRESSURE_OUTPUT);   // PID_Compact
   END_IF;
END_REGION

REGION Network 33: OUTPUT
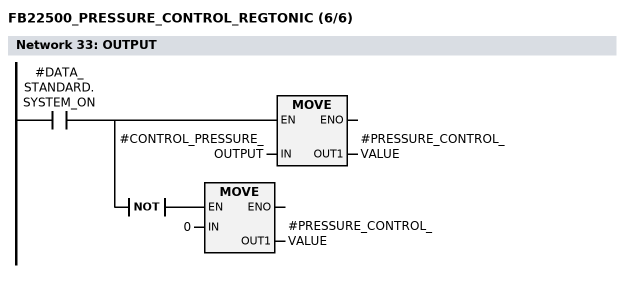
   RUNG wire#powerrail
      Contact( #DATA_STANDARD.SYSTEM_ON )
      wire#w1
      Move(in := #CONTROL_PRESSURE_OUTPUT, out1 => #PRESSURE_CONTROL_VALUE)
   END_RUNG
   RUNG wire#w1
      Not()
      Move(in := 0, out1 => #PRESSURE_CONTROL_VALUE)
   END_RUNG
   // the same network as SCL:
   IF #DATA_STANDARD.SYSTEM_ON THEN #PRESSURE_CONTROL_VALUE := #CONTROL_PRESSURE_OUTPUT; END_IF;
   IF NOT #DATA_STANDARD.SYSTEM_ON THEN #PRESSURE_CONTROL_VALUE := 0; END_IF;
END_REGION
END_FUNCTION_BLOCK
